(* IEC 61131-3 sources: POMIRTS_lab3/AS/Library/AsARCfg, 3 files *)

(* ---- AsARCfg.typ ---- *)
(********************************************************************
 * COPYRIGHT -- Bernecker + Rainer
 ********************************************************************
 * Library: AsARCfg
 * File: AsARCfg.typ
 * Author: B+R
 ********************************************************************
 * Data types of library AsARCfg
 ********************************************************************)

 TYPE
	cfgLease_typ : STRUCT				(*lease structure*)
		name			: STRING[8];	(*name of lease (max 8)*)
		startAdr		: STRING[16];	(*start address of lease*)
		stopAdr			: STRING[16];	(*stop address of lease*)
		subnetMask		: STRING[16];	(*subnet mask of lease*)
		defaultGateway	: STRING[16];	(*default gateway of lease*)
		leaseTimeout	: DINT;			(*-1 for infinite timeout*)
	END_STRUCT;
END_TYPE

(* ---- AsARCfg.fun ---- *)
(********************************************************************
 * COPYRIGHT -- Bernecker + Rainer
 ********************************************************************
 * Library: AsARCfg
 * File: AsARCfg.fun
 * Author: B+R
 ********************************************************************
 * Functions and function blocks of library AsARCfg
 ********************************************************************)

FUNCTION_BLOCK CfgGetInaNode			(*reads the node number from the AR registry for a INA device; asynchronous execution*)
	VAR_INPUT
		enable			: BOOL;			(*enables execution*)
		pDevice			: UDINT;		(*INA device name given as pointer (syntax: SL<x>.SS<y>.IF<z>)*)
	END_VAR

	VAR_OUTPUT
		status			: UINT;			(*execution status: ERR_OK, ERR_FUB_ENABLE_FALSE, ERR_FUB_BUSY, 0xXXXX = see help*)
		InaNode			: USINT;		(*INA node number*)
	END_VAR

	VAR
        i_state			: UINT;			(*internal variable*)
		i_result		: UINT;			(*internal variable*)
        i_tmp			: UDINT;		(*internal variable*)
	END_VAR
END_FUNCTION_BLOCK

FUNCTION_BLOCK CfgSetInaNode			(*enters the node number into the AR registry for INA device; asynchronous execution*)
	VAR_INPUT
		enable			: BOOL;			(*enables execution*)
		pDevice			: UDINT;		(*INA device name given as pointer (syntax: SL<x>.SS<y>.IF<z>)*)
		InaNode			: USINT;		(*INA node number*)
		Option			: UDINT;		(*options: cfgOPTION_VOLATILE, cfgOPTION_NON_VOLATILE*)
	END_VAR

	VAR_OUTPUT
		status			: UINT;			(*execution status: ERR_OK, ERR_FUB_ENABLE_FALSE, ERR_FUB_BUSY, 0xXXXX = see help*)
	END_VAR

	VAR
        i_state			: UINT;			(*internal variable*)
		i_result		: UINT;			(*internal variable*)
        i_tmp			: UDINT;		(*internal variable*)
	END_VAR
END_FUNCTION_BLOCK

FUNCTION_BLOCK CfgGetIPAddr				(*reads IP address from the AR registry for Ethernet device; asynchronous execution*)
	VAR_INPUT
		enable			: BOOL;			(*enables execution*)
		pDevice			: UDINT;		(*INA device name given as pointer (syntax: SL<x>.SS<y>.IF<z>)*)
		pIPAddr			: UDINT;		(*IP address given as a pointer*)
		Len				: USINT;		(*length of the string (pIPAddr) -> ideally, Len = 16*)
	END_VAR

	VAR_OUTPUT
		status			: UINT;			(*execution status: ERR_OK, ERR_FUB_ENABLE_FALSE, ERR_FUB_BUSY, 0xXXXX = see help*)
	END_VAR

	VAR
        i_state			: UINT;			(*internal variable*)
		i_result		: UINT;			(*internal variable*)
        i_tmp			: UDINT;		(*internal variable*)
	END_VAR
END_FUNCTION_BLOCK

FUNCTION_BLOCK CfgSetIPAddr				(*enters IP address into the AR registry for Ethernet device; asynchronous execution*)
	VAR_INPUT
		enable			: BOOL;			(*enables execution*)
		pDevice			: UDINT;		(*INA device name given as pointer (syntax: SL<x>.SS<y>.IF<z>)*)
		pIPAddr			: UDINT;		(*IP address given as pointer, valid range "1.0.0.1" - "247.255.255.255"*)
		Option			: UDINT;		(*options:  cfgOPTION_VOLATILE, cfgOPTION_NON_VOLATILE*)
	END_VAR

	VAR_OUTPUT
		status			: UINT;			(*execution status: ERR_OK, ERR_FUB_ENABLE_FALSE, ERR_FUB_BUSY, 0xXXXX = see help*)
	END_VAR

	VAR
        i_state			: UINT;			(*internal variable*)
		i_result		: UINT;			(*internal variable*)
        i_tmp			: UDINT;		(*internal variable*)
	END_VAR
END_FUNCTION_BLOCK

FUNCTION_BLOCK CfgGetSubnetMask			(*reads subnet mask from the AR registry for Ethernet device; asynchronous execution*)
	VAR_INPUT
		enable			: BOOL;			(*enables execution*)
		pDevice			: UDINT;		(*INA device name given as pointer (syntax: SL<x>.SS<y>.IF<z>)*)
		pSubnetMask		: UDINT;		(*subnet mask*)
		Len				: USINT;		(*length of the string (pSubnetMask) -> ideally, Len = 16*)
	END_VAR

	VAR_OUTPUT
		status			: UINT;			(*execution status: ERR_OK, ERR_FUB_ENABLE_FALSE, ERR_FUB_BUSY, 0xXXXX = see help*)
	END_VAR

	VAR
		i_state			: UINT;			(*internal variable*)
		i_result		: UINT;			(*internal variable*)
        i_tmp			: UDINT;		(*internal variable*)
	END_VAR
END_FUNCTION_BLOCK

FUNCTION_BLOCK CfgSetSubnetMask			(*enters subnet mask into the AR registry for Ethernet device; asynchronous execution*)
	VAR_INPUT
		enable			: BOOL;			(*enables execution*)
		pDevice			: UDINT;		(*INA device name given as pointer (syntax: SL<x>.SS<y>.IF<z>)*)
		pSubnetMask		: UDINT;		(*subnet mask given as a pointer, valid range "1.0.0.1" - "255.255.255.254"*)
		Option			: UDINT;		(*options: cfgOPTION_VOLATILE, cfgOPTION_NON_VOLATILE*)
	END_VAR

	VAR_OUTPUT
		status			: UINT;			(*execution status: ERR_OK, ERR_FUB_ENABLE_FALSE, ERR_FUB_BUSY, 0xXXXX = see help*)
	END_VAR

	VAR
        i_state			: UINT;			(*internal variable*)
		i_result		: UINT;			(*internal variable*)
        i_tmp			: UDINT;		(*internal variable*)
	END_VAR
END_FUNCTION_BLOCK

FUNCTION_BLOCK CfgGetDefaultGateway		(*reads default gateway from AR registry for Ethernet device; asynchronous execution*)
	VAR_INPUT
		enable			: BOOL;			(*enables execution*)
		pDevice			: UDINT;		(*INA device name given as pointer (syntax: SL<x>.SS<y>.IF<z>)*)
		pGateway		: UDINT;		(*default gateway address given as pointer*)
		Len				: USINT;		(*length of the string (pGateway) -> ideally, Len = 16*)
	END_VAR

	VAR_OUTPUT
		status			: UINT;			(*execution status: ERR_OK, ERR_FUB_ENABLE_FALSE, ERR_FUB_BUSY, 0xXXXX = see help*)
	END_VAR

	VAR
        i_state			: UINT;			(*internal variable*)
		i_result		: UINT;			(*internal variable*)
        i_tmp			: UDINT;		(*internal variable*)
	END_VAR
END_FUNCTION_BLOCK

FUNCTION_BLOCK CfgSetDefaultGateway		(*enters default gateway into AR registry for Ethernet device; asynchronous execution*)
	VAR_INPUT
		enable			: BOOL;			(*enables execution*)
		pDevice			: UDINT;		(*INA device name given as pointer (syntax: SL<x>.SS<y>.IF<z>)*)
		pGateway		: UDINT;		(*default gateway address given as pointer, valid range "1.0.0.1" - "247.255.255.255"*)
		Option			: UDINT;		(*options: cfgOPTION_VOLATILE, cfgOPTION_NON_VOLATILE*)
	END_VAR

	VAR_OUTPUT
		status			: UINT;			(*execution status: ERR_OK, ERR_FUB_ENABLE_FALSE, ERR_FUB_BUSY, 0xXXXX = see help*)
	END_VAR

	VAR
        i_state			: UINT;			(*internal variable*)
		i_result		: UINT;			(*internal variable*)
        i_tmp			: UDINT;		(*internal variable*)
	END_VAR
END_FUNCTION_BLOCK

FUNCTION_BLOCK CfgGetBroadcastAddr		(*reads broadcast address from AR registry for Ethernet device; asynchronous execution*)
	VAR_INPUT
		enable			: BOOL;			(*enables execution*)
		pDevice			: UDINT;		(*INA device name given as pointer (syntax: SL<x>.SS<y>.IF<z>)*)
		pBroadcastAddr	: UDINT;		(*broadcast address given as a pointer*)
		Len				: USINT;		(*length of the string (pBroadcastAddr) -> ideally, Len = 16*)
	END_VAR

	VAR_OUTPUT
		status			: UINT;			(*execution status: ERR_OK, ERR_FUB_ENABLE_FALSE, ERR_FUB_BUSY, 0xXXXX = see help*)
	END_VAR

	VAR
        i_state			: UINT;			(*internal variable*)
		i_result		: UINT;			(*internal variable*)
        i_tmp			: UDINT;		(*internal variable*)
	END_VAR
END_FUNCTION_BLOCK

FUNCTION_BLOCK CfgSetBroadcastAddr		(*enters broadcast address into the AR registry for Ethernet device; asynchronous execution*)
	VAR_INPUT
		enable			: BOOL;			(*enables execution*)
		pDevice			: UDINT;		(*INA device name given as pointer (syntax: SL<x>.SS<y>.IF<z>)*)
		pBroadcastAddr	: UDINT;		(*broadcast address given as a pointer, valid range "1.0.0.1" - "255.255.255.255"*)
		Option			: UDINT;		(*options: cfgOPTION_VOLATILE, cfgOPTION_NON_VOLATILE*)
	END_VAR

	VAR_OUTPUT
		status			: UINT;			(*execution status: ERR_OK, ERR_FUB_ENABLE_FALSE, ERR_FUB_BUSY, 0xXXXX = see help*)
	END_VAR

	VAR
        i_state			: UINT;			(*internal variable*)
		i_result		: UINT;			(*internal variable*)
        i_tmp			: UDINT;		(*internal variable*)
	END_VAR
END_FUNCTION_BLOCK

FUNCTION_BLOCK CfgGetEthBaudrate		(*reads the baud rate from the AR registry for Ethernet device; asynchronous execution*)
	VAR_INPUT
		enable			: BOOL;			(*enables execution*)
		pDevice			: UDINT;		(*INA device name given as pointer (syntax: SL<x>.SS<y>.IF<z>)*)
	END_VAR

	VAR_OUTPUT
		status			: UINT;			(*execution status: ERR_OK, ERR_FUB_ENABLE_FALSE, ERR_FUB_BUSY, 0xXXXX = see help*)
		Baudrate		: UDINT;		(*baud rate, e.g. cfgETHBAUDRATE_AUTO, cfgETHBAUDRATE_10, cfgETHBAUDRATE_10FD ...*)
	END_VAR

	VAR
        i_state			: UINT;			(*internal variable*)
		i_result		: UINT;			(*internal variable*)
        i_tmp			: UDINT;		(*internal variable*)
	END_VAR
END_FUNCTION_BLOCK

FUNCTION_BLOCK CfgSetEthBaudrate		(*enters the baud rate into the AR registry for Ethernet device; asynchronous execution*)
	VAR_INPUT
		enable			: BOOL;			(*enables execution*)
		pDevice			: UDINT;		(*INA device name given as pointer (syntax: SL<x>.SS<y>.IF<z>)*)
		Baudrate		: UDINT;		(*Ethernet baud rate, e.g. cfgETHBAUDRATE_AUTO, cfgETHBAUDRATE_10, cfgETHBAUDRATE_10FD ...*)
		Option			: UDINT;		(*options: cfgOPTION_VOLATILE, cfgOPTION_NON_VOLATILE*)
	END_VAR

	VAR_OUTPUT
		status			: UINT;			(*execution status: ERR_OK, ERR_FUB_ENABLE_FALSE, ERR_FUB_BUSY, 0xXXXX = see help*)
	END_VAR

	VAR
        i_state			: UINT;			(*internal variable*)
		i_result		: UINT;			(*internal variable*)
        i_tmp			: UDINT;		(*internal variable*)
	END_VAR
END_FUNCTION_BLOCK

FUNCTION_BLOCK CfgGetEthConfigMode		(*reads the configuration mode; asynchronous execution*)
	VAR_INPUT
		enable			: BOOL;			(*enables execution*)
		pDevice			: UDINT;		(*INA device name given as pointer (syntax: SL<x>.SS<y>.IF<z>)*)
	END_VAR

	VAR_OUTPUT
		status			: UINT;			(*execution status: ERR_OK, ERR_FUB_ENABLE_FALSE, ERR_FUB_BUSY, 0xXXXX = see help*)
		ConfigMode		: UDINT;		(*configuration mode: cfgCONFIGMODE_MANUALLY, cfgCONFIGMODE_DHCPCLIENT*)
	END_VAR

	VAR
        i_state			: UINT;			(*internal variable*)
		i_result		: UINT;			(*internal variable*)
        i_tmp			: UDINT;		(*internal variable*)
	END_VAR
END_FUNCTION_BLOCK

FUNCTION_BLOCK CfgSetEthConfigMode		(*modifies the configuration mode for Ethernet device; asynchronous execution*)
	VAR_INPUT
		enable			: BOOL;			(*enables execution*)
		pDevice			: UDINT;		(*INA device name given as pointer (syntax: SL<x>.SS<y>.IF<z>)*)
		ConfigMode		: UDINT;		(*configuration mode: cfgCONFIGMODE_MANUALLY, cfgCONFIGMODE_DHCPCLIENT*)
		Option			: UDINT;		(*options: cfgOPTION_VOLATILE, cfgOPTION_NON_VOLATILE*)
	END_VAR

	VAR_OUTPUT
		status			: UINT;			(*execution status: ERR_OK, ERR_FUB_ENABLE_FALSE, ERR_FUB_BUSY, 0xXXXX = see help*)
	END_VAR

	VAR
        i_state			: UINT;			(*internal variable*)
		i_result		: UINT;			(*internal variable*)
        i_tmp			: UDINT;		(*internal variable*)
	END_VAR
END_FUNCTION_BLOCK

FUNCTION_BLOCK CfgGetHostName			(*reads a host name for a target; asynchronous execution*)
	VAR_INPUT
		enable			: BOOL;			(*enables execution*)
		pHostName		: UDINT;		(*hostname*)
		Len				: USINT;		(*length of the string (HostName)*)
	END_VAR

	VAR_OUTPUT
		status			: UINT;			(*execution status: ERR_OK, ERR_FUB_ENABLE_FALSE, ERR_FUB_BUSY, 0xXXXX = see help*)
	END_VAR

	VAR
        i_state			: UINT;			(*internal variable*)
		i_result		: UINT;			(*internal variable*)
        i_tmp			: UDINT;		(*internal variable*)
	END_VAR
END_FUNCTION_BLOCK

FUNCTION_BLOCK CfgSetHostName			(*sets a host name for a target; asynchronous execution*)
	VAR_INPUT
		enable			: BOOL;			(*enables execution*)
		pHostName		: UDINT;		(*hostname*)
		Option			: UDINT;		(*options: cfgOPTION_VOLATILE, cfgOPTION_NON_VOLATILE*)
	END_VAR

	VAR_OUTPUT
		status			: UINT;			(*execution status: ERR_OK, ERR_FUB_ENABLE_FALSE, ERR_FUB_BUSY, 0xXXXX = see help*)
	END_VAR

	VAR
        i_state			: UINT;			(*internal variable*)
		i_result		: UINT;			(*internal variable*)
        i_tmp			: UDINT;		(*internal variable*)
	END_VAR
END_FUNCTION_BLOCK

FUNCTION_BLOCK CfgGetMacAddr			(*reads the MAC address of an Ethernet device*)
	VAR_INPUT
		enable			: BOOL;			(*enables execution*)
		pDevice			: UDINT;		(*INA device name given as pointer (syntax: SL<x>.SS<y>.IF<z>)*)
		pMacAddr		: UDINT;		(*MAC address (pointer to buffer where the MAC address should be written)*)
		Len				: USINT;		(*length of the MAC address (buffer - pMacAddr) -> normally 6 bytes*)
	END_VAR

	VAR_OUTPUT
		status			: UINT;			(*execution status: ERR_OK, ERR_FUB_ENABLE_FALSE, 0xXXXX = see help*)
	END_VAR

	VAR
        i_state			: UINT;			(*internal variable*)
		i_result		: UINT;			(*internal variable*)
        i_tmp			: UDINT;		(*internal variable*)
	END_VAR
END_FUNCTION_BLOCK

FUNCTION_BLOCK CfgSetFTPServer			(*enables/disables the FTP server*)
	VAR_INPUT
		enable			: BOOL;			(*enables execution*)
		Option			: UDINT;		(*options: cfgOPTION_DISABLE, cfgOPTION_ENABLE*)
	END_VAR

	VAR_OUTPUT
		status			: UINT;			(*execution status: ERR_OK, ERR_FUB_ENABLE_FALSE, 0xXXXX = see help*)
	END_VAR

	VAR
        i_state			: UINT;			(*internal variable*)
		i_result		: UINT;			(*internal variable*)
        i_tmp			: UDINT;		(*internal variable*)
	END_VAR
END_FUNCTION_BLOCK

FUNCTION_BLOCK CfgGetTimeOffset			(*returns the configured time offset*)
	VAR_INPUT
		enable			: BOOL;			(*enables execution*)
	END_VAR

	VAR_OUTPUT
		status			: UINT;			(*execution status: ERR_OK, ERR_FUB_ENABLE_FALSE, 0xXXXX = see help*)
		timeoffset		: INT;			(*configured time offset*)
	END_VAR

	VAR
        i_state			: UINT;			(*internal variable*)
		i_result		: UINT;			(*internal variable*)
        i_tmp			: UDINT;		(*internal variable*)
	END_VAR
END_FUNCTION_BLOCK

FUNCTION_BLOCK CfgSetTimeOffset			(*sets a time offset*)
	VAR_INPUT
		enable			: BOOL;			(*enables execution*)
        timeoffset		: INT;			(*configured time offset*)
        option			: UDINT;		(*options: cfgOPTION_VOLATILE, cfgOPTION_NON_VOLATILE*)
	END_VAR

	VAR_OUTPUT
        status			: UINT;			(*execution status: ERR_OK, ERR_FUB_ENABLE_FALSE, 0xXXXX = see help*)
	END_VAR

	VAR
        i_state			: UINT;			(*internal variable*)
		i_result		: UINT;			(*internal variable*)
        i_tmp			: UDINT;		(*internal variable*)
	END_VAR
END_FUNCTION_BLOCK

FUNCTION_BLOCK CfgSetSntpServer			(*starts the SNTP server*)
	VAR_INPUT
		enable			: BOOL;			(*enables execution*)
        start			: UDINT;		(*1 Starts the SNTP server*)
        option			: UDINT;		(*Options: cfgOPTION_VOLATILE, cfgOPTION_NON_VOLATILE*)
	END_VAR

	VAR_OUTPUT
        status			: UINT;			(*execution status: ERR_OK, ERR_FUB_ENABLE_FALSE, 0xXXXX = see help*)
	END_VAR

	VAR
        i_state			: UINT;			(*internal variable*)
		i_result		: UINT;			(*internal variable*)
        i_tmp			: UDINT;		(*internal variable*)
	END_VAR
END_FUNCTION_BLOCK

FUNCTION_BLOCK CfgSetSntpClient			(*starts and stops the SNTP client*)
	VAR_INPUT
		enable			: BOOL;			(*enables execution*)
		run				: UDINT;		(*0 stop client, 1 start client*)
		pServerAddr		: UDINT;		(*pointer to a string with the IP address of the SNTP server*)
		sntpcInterval	: UINT;			(*interval in minutes that it takes for the SNTP client to synchronize the time with the server*)
		rtcInterval		: UINT;			(*interval in minutes that it takes to synchronize the RTC with the software time during SNTP operation*)
		option			: UDINT;		(*options: cfgOPTION_VOLATILE, cfgOPTION_NON_VOLATILE*)
	END_VAR

	VAR_OUTPUT
		status			: UINT;			(*execution status: ERR_OK, ERR_FUB_ENABLE_FALSE, 0xXXXX = see help*)
		syncStatus		: USINT;		(*0 Client not active, 1 Client already active, but time not received from server, ...*)
	END_VAR

	VAR
        i_state			: UINT;			(*internal variable*)
		i_result		: UINT;			(*internal variable*)
        i_tmp			: UDINT;		(*internal variable*)
	END_VAR
END_FUNCTION_BLOCK

FUNCTION_BLOCK CfgGetSntpcData			(*returns the parameters relevant for the SNTP client*)
	VAR_INPUT
		enable			: BOOL;			(*enables execution*)
		pServerAddr		: UDINT;		(*pointer to a long enough string to contain the server address or server name*)
		Len				: USINT;		(*length of the string (pServerAddr)*)
	END_VAR

	VAR_OUTPUT
		status			: UINT;			(*execution status: ERR_OK, ERR_FUB_ENABLE_FALSE, 0xXXXX = see help*)
		run				: UDINT;		(*1 Client active, 0 Client inactive*)
        sntpcInterval	: UINT;			(*interval that it takes for the SNTP client to synchronize the time with the server*)
        rtcInterval		: UINT;			(*interval that it take to synchronize the RTC with the software time during SNTP operation*)
	END_VAR

	VAR
        i_state			: UINT;			(*internal variable*)
		i_result		: UINT;			(*internal variable*)
        i_tmp			: UDINT;		(*internal variable*)
	END_VAR
END_FUNCTION_BLOCK

FUNCTION_BLOCK CfgGetSntpsData			(*returns whether the SNTP server is active*)
	VAR_INPUT
		enable			: BOOL;			(*enables execution*)
	END_VAR

	VAR_OUTPUT
		status			: UINT;			(*execution status: ERR_OK, ERR_FUB_ENABLE_FALSE, 0xXXXX = see help*)
		run				: UDINT;		(*1 server active, 0 server inactive*)
	END_VAR

	VAR
        i_state			: UINT;			(*internal variable*)
		i_result		: UINT;			(*internal variable*)
        i_tmp			: UDINT;		(*internal variable*)
	END_VAR
END_FUNCTION_BLOCK

FUNCTION_BLOCK CfgGetTimeZone
	VAR_INPUT
		enable			: BOOL;			(*enables execution*)
	END_VAR

	VAR_OUTPUT
		timezoneID		: UINT;
        status			: UINT;			(*execution status: ERR_OK, ERR_FUB_ENABLE_FALSE, ERR_FUB_BUSY, 0xXXXX = see help*)
	END_VAR

	VAR
        i_state			: UINT;			(*internal variable*)
		i_result		: UINT;			(*internal variable*)
        i_tmp			: UDINT;		(*internal variable*)
	END_VAR
END_FUNCTION_BLOCK

FUNCTION_BLOCK CfgSetTimeZone
	VAR_INPUT
		enable			: BOOL;			(*enables execution*)
		timezoneID		: UINT;
		option			: UDINT;
	END_VAR

	VAR_OUTPUT
        status			: UINT;			(*execution status: ERR_OK, ERR_FUB_ENABLE_FALSE, ERR_FUB_BUSY, 0xXXXX = see help*)
	END_VAR

	VAR
        i_state			: UINT;			(*internal variable*)
		i_result		: UINT;			(*internal variable*)
        i_tmp			: UDINT;		(*internal variable*)
	END_VAR
END_FUNCTION_BLOCK

FUNCTION_BLOCK CfgGetTimeZoneInfo
	VAR_INPUT
		enable			: BOOL;			(*enables execution*)
		timezoneID		: UINT;
	END_VAR

	VAR_OUTPUT
		gmt				: INT;
		gmtDst			: INT;
        status			: UINT;			(*execution status: ERR_OK, ERR_FUB_ENABLE_FALSE, ERR_FUB_BUSY, 0xXXXX = see help*)
	END_VAR

	VAR
        i_state			: UINT;			(*internal variable*)
		i_result		: UINT;			(*internal variable*)
        i_tmp			: UDINT;		(*internal variable*)
	END_VAR
END_FUNCTION_BLOCK

FUNCTION_BLOCK CfgGetTimeZoneEntry
	VAR_INPUT
		enable			: BOOL;			(*enables execution*)
		timezoneID		: UINT;
		year			: UINT;
	END_VAR

	VAR_OUTPUT
		dateDst			: DATE_AND_TIME;
		dateNormal		: DATE_AND_TIME;
        status			: UINT;			(*execution status: ERR_OK, ERR_FUB_ENABLE_FALSE, ERR_FUB_BUSY, 0xXXXX = see help*)
	END_VAR

	VAR
        i_state			: UINT;			(*internal variable*)
		i_result		: UINT;			(*internal variable*)
        i_tmp			: UDINT;		(*internal variable*)
	END_VAR
END_FUNCTION_BLOCK

FUNCTION_BLOCK CfgGetDst
	VAR_INPUT
		enable			: BOOL;			(*enables execution*)
	END_VAR

	VAR_OUTPUT
		dst				: BOOL;
        status			: UINT;			(*execution status: ERR_OK, ERR_FUB_ENABLE_FALSE, ERR_FUB_BUSY, 0xXXXX = see help*)
	END_VAR

	VAR
        i_state			: UINT;			(*internal variable*)
		i_result		: UINT;			(*internal variable*)
        i_tmp			: UDINT;		(*internal variable*)
	END_VAR
END_FUNCTION_BLOCK

FUNCTION_BLOCK CfgSetDst
	VAR_INPUT
		enable			: BOOL;			(*enables execution*)
		dst				: BOOL;
		option			: UDINT;
	END_VAR

	VAR_OUTPUT
        status			: UINT;			(*execution status: ERR_OK, ERR_FUB_ENABLE_FALSE, ERR_FUB_BUSY, 0xXXXX = see help*)
	END_VAR

	VAR
        i_state			: UINT;			(*internal variable*)
		i_result		: UINT;			(*internal variable*)
        i_tmp			: UDINT;		(*internal variable*)
	END_VAR
END_FUNCTION_BLOCK

FUNCTION_BLOCK CfgGetCIFSDomain				(*cifs - reads domain name from the AR registry; asynchronous execution*)
	VAR_INPUT
		enable			: BOOL;			(*enables execution*)
		pDomain			: UDINT;		(*Domainname given as a pointer*)
		Len				: USINT;		(*length of the string (pDomain) -> ideally, Len = 16*)
	END_VAR

	VAR_OUTPUT
		isWorkgroup		: USINT;		(*specifies if Workgroup or Domain*)
		status			: UINT;			(*execution status: ERR_OK, ERR_FUB_ENABLE_FALSE, ERR_FUB_BUSY, 0xXXXX = see help*)
	END_VAR

	VAR
        i_state			: UINT;			(*internal variable*)
		i_result		: UINT;			(*internal variable*)
        i_tmp			: UDINT;		(*internal variable*)
	END_VAR
END_FUNCTION_BLOCK

FUNCTION_BLOCK CfgSetCIFSDomain			(*cifs - enters domain into the AR registry; asynchronous execution*)
	VAR_INPUT
		enable			: BOOL;			(*enables execution*)
		pDomain			: UDINT;		(*Domainname given as pointer*)
		isWorkgroup		: USINT;		(*specifies if Workgroup or Domain cfgOPTION_NON_WORKGROUP, cfgOPTION_WORKGROUP*)
		Option			: UDINT;		(*options:  cfgOPTION_VOLATILE, cfgOPTION_NON_VOLATILE*)
	END_VAR

	VAR_OUTPUT
		status			: UINT;			(*execution status: ERR_OK, ERR_FUB_ENABLE_FALSE, ERR_FUB_BUSY, 0xXXXX = see help*)
	END_VAR

	VAR
        i_state			: UINT;			(*internal variable*)
		i_result		: UINT;			(*internal variable*)
        i_tmp			: UDINT;		(*internal variable*)
	END_VAR
END_FUNCTION_BLOCK

FUNCTION_BLOCK CfgGetCIFSDefaultuser	(*cifs - reads default user from the AR registry; asynchronous execution*)
	VAR_INPUT
		enable				: BOOL;			(*enables execution*)
		pDefaultuser		: UDINT;		(*Default Username given as a pointer*)
		lenUser				: USINT;		(*length of the string (pDefaultuser) -> ideally, Len = 16*)
		pDefaultpassword	: UDINT;		(*Default Password given as a pointer*)
		lenPassword			: USINT;		(*length of the string (pDefaultpassword) -> ideally, Len = 16*)
	END_VAR

	VAR_OUTPUT
		status			: UINT;			(*execution status: ERR_OK, ERR_FUB_ENABLE_FALSE, ERR_FUB_BUSY, 0xXXXX = see help*)
	END_VAR

	VAR
        i_state			: UINT;			(*internal variable*)
		i_result		: UINT;			(*internal variable*)
        i_tmp			: UDINT;		(*internal variable*)
	END_VAR
END_FUNCTION_BLOCK

FUNCTION_BLOCK CfgSetCIFSDefaultuser	(*cifs - enters default user into the AR registry; asynchronous execution*)
	VAR_INPUT
		enable				: BOOL;			(*enables execution*)
		pDefaultuser		: UDINT;		(*Default Username given as pointer*)
		pDefaultpassword	: UDINT;		(*Default Password given as a pointer*)
		Option				: UDINT;		(*options:  cfgOPTION_VOLATILE, cfgOPTION_NON_VOLATILE*)
	END_VAR

	VAR_OUTPUT
		status			: UINT;			(*execution status: ERR_OK, ERR_FUB_ENABLE_FALSE, ERR_FUB_BUSY, 0xXXXX = see help*)
	END_VAR

	VAR
        i_state			: UINT;			(*internal variable*)
		i_result		: UINT;			(*internal variable*)
        i_tmp			: UDINT;		(*internal variable*)
	END_VAR
END_FUNCTION_BLOCK

FUNCTION_BLOCK CfgSetDhcpServer 	(*dhcp - starts or stops dhcp server*)
	VAR_INPUT
		enable				: BOOL;			(*enables execution*)
		start				: UDINT;		(*1 = start server; 0 = stop server*)
		option				: UDINT;		(*options:  cfgOPTION_VOLATILE, cfgOPTION_NON_VOLATILE*)
	END_VAR

	VAR_OUTPUT
		status			: UINT;			(*execution status: ERR_OK, ERR_FUB_ENABLE_FALSE, ERR_FUB_BUSY, 0xXXXX = see help*)
	END_VAR

	VAR
        i_state			: UINT;			(*internal variable*)
		i_result		: UINT;			(*internal variable*)
        i_tmp			: UDINT;		(*internal variable*)
	END_VAR
END_FUNCTION_BLOCK

FUNCTION_BLOCK CfgSetDhcpsData 	(*dhcp - configures dhcp server*)
	VAR_INPUT
		enable				: BOOL;			(*enables execution*)
		pInterfaceList		: UDINT;		(*provided interfaces*)
		pLeases				: UDINT;		(*provided leases*)
		numLeases			: UDINT;		(*number of leases*)
		option				: UDINT;		(*options:  cfgOPTION_VOLATILE, cfgOPTION_NON_VOLATILE*)
	END_VAR

	VAR_OUTPUT
		status			: UINT;			(*execution status: ERR_OK, ERR_FUB_ENABLE_FALSE, ERR_FUB_BUSY, 0xXXXX = see help*)
	END_VAR

	VAR
        i_state			: UINT;			(*internal variable*)
		i_result		: UINT;			(*internal variable*)
        i_tmp			: UDINT;		(*internal variable*)
	END_VAR
END_FUNCTION_BLOCK

FUNCTION_BLOCK CfgGetDhcpsData 	(*dhcp - reads configuration of dhcp server*)
	VAR_INPUT
		enable				: BOOL;			(*enables execution*)
		pInterfaceList		: UDINT;		(*provided interfaces*)
		len					: UDINT;		(*length of the string (pInterfaces)*)
		pLeases				: UDINT;		(*provided leases*)
		numLeases			: UDINT;		(*number of leases*)
	END_VAR

	VAR_OUTPUT
		startMode		: UDINT;		(*1 = server is working; 0 = server is not working*)
		numNeeded		: UDINT;		(*needed length*)
		status			: UINT;			(*execution status: ERR_OK, ERR_FUB_ENABLE_FALSE, ERR_FUB_BUSY, 0xXXXX = see help*)
	END_VAR

	VAR
        i_state			: UINT;			(*internal variable*)
		i_result		: UINT;			(*internal variable*)
        i_tmp			: UDINT;		(*internal variable*)
	END_VAR
END_FUNCTION_BLOCK

FUNCTION_BLOCK CfgSetSdmStatus			(*enables/disables data refresh of system diagnostics manager*)
	VAR_INPUT
		enable			: BOOL;			(*enables execution*)
		start			: UDINT;		(*options: cfgOPTION_ENABLE_SDM; cfgOPTION_DISABLE_SDM*)
		Option			: UDINT;		(*reserve*)
	END_VAR

	VAR_OUTPUT
		status			: UINT;			(*execution status: ERR_OK, ERR_FUB_ENABLE_FALSE, 0xXXXX = see help*)
	END_VAR

	VAR
        i_state			: UINT;			(*internal variable*)
		i_result		: UINT;			(*internal variable*)
        i_tmp			: UDINT;		(*internal variable*)
	END_VAR
END_FUNCTION_BLOCK

FUNCTION_BLOCK CfgGetSdmStatus			(*returns whether the system diagnostics manager is active*)
	VAR_INPUT
		enable			: BOOL;			(*enables execution*)
	END_VAR

	VAR_OUTPUT
		status			: UINT;			(*execution status: ERR_OK, ERR_FUB_ENABLE_FALSE, 0xXXXX = see help*)
		run				: UDINT;		(*status: cfgSTATUS_SDM_ENABLED, cfgSTATUS_SDM_DISABLED*)
	END_VAR

	VAR
        i_state			: UINT;			(*internal variable*)
		i_result		: UINT;			(*internal variable*)
        i_tmp			: UDINT;		(*internal variable*)
	END_VAR
END_FUNCTION_BLOCK

FUNCTION CfgClearNV		: UINT			(*clear non volatile data*)
END_FUNCTION

FUNCTION_BLOCK CfgSetSdmColor			(*set the system diagnostics manager color scheme*)
	VAR_INPUT
		enable			: BOOL;			(*enables execution*)
		red  			: UDINT;  		(*red value (0-255)*)
		green  			: UDINT;  		(*green value (0-255)*)
		blue  			: UDINT;  		(*blue value (0-255)*)
		Option			: UDINT;		(*options: cfgOPTION_VOLATILE, cfgOPTION_NON_VOLATILE*)
	END_VAR

	VAR_OUTPUT
		status			: UINT;			(*execution status: ERR_OK, ERR_FUB_ENABLE_FALSE, 0xXXXX = see help*)
	END_VAR

	VAR
        i_state			: UINT;			(*internal variable*)
		i_result		: UINT;			(*internal variable*)
        i_tmp			: UDINT;		(*internal variable*)
	END_VAR
END_FUNCTION_BLOCK

FUNCTION_BLOCK CfgGetSdmColor			(*get the system diagnostics manager color scheme*)
	VAR_INPUT
		enable			: BOOL;			(*enables execution*)
	END_VAR

	VAR_OUTPUT
		status			: UINT;			(*execution status: ERR_OK, ERR_FUB_ENABLE_FALSE, 0xXXXX = see help*)
		red  			: UDINT;  		(*red value (0-255)*)
		green  			: UDINT;  		(*green value (0-255)*)
		blue  			: UDINT;  		(*blue value (0-255)*)
	END_VAR

	VAR
        i_state			: UINT;			(*internal variable*)
		i_result		: UINT;			(*internal variable*)
        i_tmp			: UDINT;		(*internal variable*)
	END_VAR
END_FUNCTION_BLOCK

FUNCTION_BLOCK CfgGetSdmCustomData1 	(*sdm - get custom data 1 *)
	VAR_INPUT
		enable			: BOOL;			(*enables execution*)
		pDevice			: UDINT;		(*Devicename given as a pointer*)
		lenDevice		: UDINT;		(*length of the string (pDevice) -> ideally, Len = 255*)
		pFile			: UDINT;		(*Filename given as a pointer*)
		lenFile			: UDINT;		(*length of the string (pFile) -> ideally, Len = 255*)
		pDatamodule		: UDINT;		(*Datamodulename given as a pointer*)
		lenDatamodule	: UDINT;		(*length of the string (pDatamodule) -> ideally, Len = 255*)
	END_VAR

	VAR_OUTPUT
		status			: UINT;			(*execution status: ERR_OK, ERR_FUB_ENABLE_FALSE, ERR_FUB_BUSY, 0xXXXX = see help*)
	END_VAR

	VAR
        i_state			: UINT;			(*internal variable*)
		i_result		: UINT;			(*internal variable*)
        i_tmp			: UDINT;		(*internal variable*)
	END_VAR
END_FUNCTION_BLOCK

FUNCTION_BLOCK CfgSetSdmCustomData1 	(*sdm - set custom data 1 *)
	VAR_INPUT
		enable			: BOOL;			(*enables execution*)
		pDevice			: UDINT;		(*Devicename given as a pointer*)
		pFile			: UDINT;		(*Filename given as a pointer*)
		pDatamodule		: UDINT;		(*Datamodulename given as a pointer*)
		Option			: UDINT;		(*options: cfgOPTION_VOLATILE, cfgOPTION_NON_VOLATILE*)
	END_VAR

	VAR_OUTPUT
		status			: UINT;			(*execution status: ERR_OK, ERR_FUB_ENABLE_FALSE, ERR_FUB_BUSY, 0xXXXX = see help*)
	END_VAR

	VAR
        i_state			: UINT;			(*internal variable*)
		i_result		: UINT;			(*internal variable*)
        i_tmp			: UDINT;		(*internal variable*)
	END_VAR
END_FUNCTION_BLOCK

FUNCTION_BLOCK CfgGetSdmCustomData2 	(*sdm - get custom data 2 *)
	VAR_INPUT
		enable			: BOOL;			(*enables execution*)
		pDevice			: UDINT;		(*Devicename given as a pointer*)
		lenDevice		: UDINT;		(*length of the string (pDevice) -> ideally, Len = 255*)
		pFile			: UDINT;		(*Filename given as a pointer*)
		lenFile			: UDINT;		(*length of the string (pFile) -> ideally, Len = 255*)
		pDatamodule		: UDINT;		(*Datamodulename given as a pointer*)
		lenDatamodule	: UDINT;		(*length of the string (pDatamodule) -> ideally, Len = 255*)
	END_VAR

	VAR_OUTPUT
		status			: UINT;			(*execution status: ERR_OK, ERR_FUB_ENABLE_FALSE, ERR_FUB_BUSY, 0xXXXX = see help*)
	END_VAR

	VAR
        i_state			: UINT;			(*internal variable*)
		i_result		: UINT;			(*internal variable*)
        i_tmp			: UDINT;		(*internal variable*)
	END_VAR
END_FUNCTION_BLOCK

FUNCTION_BLOCK CfgSetSdmCustomData2 	(*sdm - set custom data 2 *)
	VAR_INPUT
		enable			: BOOL;			(*enables execution*)
		pDevice			: UDINT;		(*Devicename given as a pointer*)
		pFile			: UDINT;		(*Filename given as a pointer*)
		pDatamodule		: UDINT;		(*Datamodulename given as a pointer*)
		Option			: UDINT;		(*options: cfgOPTION_VOLATILE, cfgOPTION_NON_VOLATILE*)
	END_VAR

	VAR_OUTPUT
		status			: UINT;			(*execution status: ERR_OK, ERR_FUB_ENABLE_FALSE, ERR_FUB_BUSY, 0xXXXX = see help*)
	END_VAR

	VAR
        i_state			: UINT;			(*internal variable*)
		i_result		: UINT;			(*internal variable*)
        i_tmp			: UDINT;		(*internal variable*)
	END_VAR
END_FUNCTION_BLOCK

FUNCTION_BLOCK CfgGetWebMimeType 	(*webserver - set mime type *)
	VAR_INPUT
		enable			: BOOL;			(*enables execution*)
		pFileExtension	: UDINT;		(*Fileextension gives a pointer*)
		pMimeType		: UDINT;		(*MimeType given as a pointer*)
		len				: UDINT;		(*length of the string (pMimeType) -> ideally, Len = 255*)
	END_VAR

	VAR_OUTPUT
		status			: UINT;			(*execution status: ERR_OK, ERR_FUB_ENABLE_FALSE, ERR_FUB_BUSY, 0xXXXX = see help*)
	END_VAR

	VAR
        i_state			: UINT;			(*internal variable*)
		i_result		: UINT;			(*internal variable*)
        i_tmp			: UDINT;		(*internal variable*)
	END_VAR
END_FUNCTION_BLOCK

FUNCTION_BLOCK CfgSetWebMimeType 	(*webserver - get mime type*)
	VAR_INPUT
		enable			: BOOL;			(*enables execution*)
		mode			: BOOL;			(*cfgWEB_MODE_MIME_DEL(0) or cfgWEB_MODE_MIME_ADD(1)*)
		pFileExtension	: UDINT;		(*Fileextension gives a pointer*)
		pMimeType		: UDINT;		(*MimeType given as a pointer*)
		Option			: UDINT;		(*options: cfgOPTION_VOLATILE, cfgOPTION_NON_VOLATILE*)
	END_VAR

	VAR_OUTPUT
		status			: UINT;			(*execution status: ERR_OK, ERR_FUB_ENABLE_FALSE, ERR_FUB_BUSY, 0xXXXX = see help*)
	END_VAR

	VAR
        i_state			: UINT;			(*internal variable*)
		i_result		: UINT;			(*internal variable*)
        i_tmp			: UDINT;		(*internal variable*)
	END_VAR
END_FUNCTION_BLOCK

FUNCTION_BLOCK CfgGetWebServerPort 	(*webserver - get port number*)
	VAR_INPUT
		enable			: BOOL;			(*enables execution*)
	END_VAR

	VAR_OUTPUT
		status			: UINT;			(*execution status: ERR_OK, ERR_FUB_ENABLE_FALSE, ERR_FUB_BUSY, 0xXXXX = see help*)
		port  			: UINT;  		(*port number*)
	END_VAR

	VAR
        i_state			: UINT;			(*internal variable*)
		i_result		: UINT;			(*internal variable*)
        i_tmp			: UDINT;		(*internal variable*)
	END_VAR
END_FUNCTION_BLOCK

FUNCTION_BLOCK CfgGetWebServerDevice 	(*webserver - get webserver root directory*)
	VAR_INPUT
		enable			: BOOL;			(*enables execution*)
		pDevice 		: UDINT;  		(*Root directory name given as pointer*)
		len				: UDINT;		(*length of the string (pDevice) -> ideally, Len = 255*)
	END_VAR

	VAR_OUTPUT
		status			: UINT;			(*execution status: ERR_OK, ERR_FUB_ENABLE_FALSE, ERR_FUB_BUSY, 0xXXXX = see help*)
	END_VAR

	VAR
        i_state			: UINT;			(*internal variable*)
		i_result		: UINT;			(*internal variable*)
        i_tmp			: UDINT;		(*internal variable*)
	END_VAR
END_FUNCTION_BLOCK

FUNCTION_BLOCK CfgGetWebAspGoform 	(*webserver - get webserver ASP form*)
	VAR_INPUT
		enable			: BOOL;			(*enables execution*)
	END_VAR

	VAR_OUTPUT
		status			: UINT;			(*execution status: ERR_OK, ERR_FUB_ENABLE_FALSE, ERR_FUB_BUSY, 0xXXXX = see help*)
		mode			: UINT;			(*webserver - get webserver ASP form*)
	END_VAR

	VAR
        i_state			: UINT;			(*internal variable*)
		i_result		: UINT;			(*internal variable*)
        i_tmp			: UDINT;		(*internal variable*)
	END_VAR
END_FUNCTION_BLOCK

FUNCTION_BLOCK CfgSetWebAspGoform 	(*webserver - set webserver ASP form*)
	VAR_INPUT
		enable			: BOOL;			(*enables execution*)
		mode			: UINT;			(*webserver - set webserver ASP form*)
		Option			: UDINT;		(*options: cfgOPTION_VOLATILE, cfgOPTION_NON_VOLATILE*)
	END_VAR

	VAR_OUTPUT
		status			: UINT;			(*execution status: ERR_OK, ERR_FUB_ENABLE_FALSE, ERR_FUB_BUSY, 0xXXXX = see help*)
	END_VAR

	VAR
        i_state			: UINT;			(*internal variable*)
		i_result		: UINT;			(*internal variable*)
        i_tmp			: UDINT;		(*internal variable*)
	END_VAR
END_FUNCTION_BLOCK

FUNCTION_BLOCK CfgGetWebServerStatus 	(*webserver - get webserver status*)
	VAR_INPUT
		enable			: BOOL;			(*enables execution*)
	END_VAR

	VAR_OUTPUT
		status			: UINT;			(*execution status: ERR_OK, ERR_FUB_ENABLE_FALSE, ERR_FUB_BUSY, 0xXXXX = see help*)
		mode			: UINT;			(*cfgWEB_MODE_DISABLED(0) cfgWEB_MODE_ENABLED(1)*)
	END_VAR

	VAR
        i_state			: UINT;			(*internal variable*)
		i_result		: UINT;			(*internal variable*)
        i_tmp			: UDINT;		(*internal variable*)
	END_VAR
END_FUNCTION_BLOCK

FUNCTION_BLOCK CfgSetWebServerStatus 	(*webserver - set webserver status*)
	VAR_INPUT
		enable			: BOOL;			(*enables execution*)
		mode			: UINT;			(*cfgWEB_MODE_DISABLED(0) cfgWEB_MODE_ENABLED(1)*)
		Option			: UDINT;		(*options: cfgOPTION_VOLATILE, cfgOPTION_NON_VOLATILE*)
	END_VAR

	VAR_OUTPUT
		status			: UINT;			(*execution status: ERR_OK, ERR_FUB_ENABLE_FALSE, ERR_FUB_BUSY, 0xXXXX = see help*)
	END_VAR

	VAR
        i_state			: UINT;			(*internal variable*)
		i_result		: UINT;			(*internal variable*)
        i_tmp			: UDINT;		(*internal variable*)
	END_VAR
END_FUNCTION_BLOCK

(* ---- AsARCfg.var ---- *)
(********************************************************************
 * COPYRIGHT -- Bernecker + Rainer
 ********************************************************************
 * Library: AsARCfg
 * File: AsARCfg.var
 * Author: B+R
 ********************************************************************
 * Local variables of library AsARCfg
 ********************************************************************)

VAR CONSTANT
	cfgERR_DEVICE_NOT_EXIST			: UINT		:= 29000;	(*device doesn't exist or device not configured*)
	cfgERR_DEVICE_INVALID			: UINT		:= 29001;	(*FBK "pDevice" parameter invalid (e.g. pDevice = 0)*)
	cfgERR_OPTION_INVALID			: UINT		:= 29002;	(*FBK "Option" parameter invalid*)
	cfgERR_VALUE_INVALID			: UINT		:= 29003;	(*invalid FBK parameter, error text depends on the function block*)
	cfgERR_SET_NOT_POSSIBLE			: UINT		:= 29004;	(*not possible to set the subnet mask (e.g. DHCP client)*)
	cfgERR_ARREG					: UINT		:= 29005;	(*error in the AR registry*)
	cfgERR_INANODE_NOT_SUPPORTED	: UINT		:= 29006;	(*INA device does not support INA node numbers (e.g. IF1 = RS232)*)
	cfgERR_FTP_SINIT				: UINT		:= 29007;	(*initialization error on FTP server*)
	cfgERR_FTP_SDOWN				: UINT		:= 29008;	(*shutdown error on FTP server*)
	cfgERR_PARAM_NOT_SET			: UINT		:= 29009;	(*default gateway not defined*)
	cfgERR_SNTP_SERVER 				: UINT		:= 29010;	(*could not start the SNTP server*)
	cfgERR_SNTP_CLIENT 				: UINT		:= 29011;	(*error starting SNTP client (e.g. client already running)*)
	cfgERR_SNTP_INTERVAL 			: UINT		:= 29012;	(*invalid FBK parameter - values from 1 to 60 are valid*)
	cfgERR_SYSTEM		 			: UINT		:= 29013;	(*unexpected system error*)
	cfgERR_TIMEZONE					: UINT		:= 29014;   (*invalid timezone specified*)
	cfgERR_YEAR_INVALID				: UINT		:= 29015;	(*invalid year specified*)
	cfgERR_CIFS_DOMAIN_INVALID		: UINT 		:= 29016;   (*cifs domain name not defined *)
	cfgERR_CIFS_DEFAULTUSER_INVALID	: UINT		:= 29017;	(*cifs defaultuser not defined *)
	cfgERR_INANODE_NUMBER_SET       : UINT      := 29018;	(*could not set the INA node number*)
	cfgERR_CIFS_DEFAULTPW_INVALID	: UINT		:= 29019;	(*cifs default password not defined *)
	cfgERR_DHCP_SERVER_STARTED		: UINT		:= 29020;	(*server is already working*)
	cfgERR_INTERFACELIST_BUFFER		: UINT		:= 29021;	(*interfacelist buffer to small*)
	cfgERR_LEASES_BUFFER			: UINT		:= 29022;	(*leases array to small*)
	cfgERR_LEASE_EXISTS				: UINT		:= 29023;	(*leasename already exists*)
	cfgERR_LEASE_TIMEOUT			: UINT		:= 29024;	(*invalid lease timeout*)
	cfgERR_SDM_FUNCTION_NOT_FOUND	: UINT		:= 29026;	(*used arsdm function was not found*)
	cfgERR_CLEAR_NV_DATA			: UINT		:= 29027;	(*could not clear NV data*)
	cfgERR_FUNCTION_NOT_FOUND	    : UINT		:= 29028;	(*referenced function was not found*)
	cfgERR_SDM_DISABLED 		    : UINT      := 29029;	(*System diagnostics disabled*)
	cfgERR_WEBSERV_DISABLED 		: UINT      := 29030;	(*Web Server disabled*)

	cfgETHBAUDRATE_AUTO				: UDINT		:= 0;		(*auto-detect*)
	cfgETHBAUDRATE_10				: UDINT		:= 10;		(*10 MBaud, half-duplex*)
	cfgETHBAUDRATE_10FD				: UDINT		:= 11;		(*10 MBaud, full-duplex*)
	cfgETHBAUDRATE_100				: UDINT		:= 100;		(*100 MBaud, half-duplex*)
	cfgETHBAUDRATE_100FD			: UDINT		:= 101;		(*100 MBaud, full-duplex*)
	cfgETHBAUDRATE_1000FD			: UDINT		:= 1001;	(*1 GBaud, full-duplex*)

	cfgOPTION_NON_VOLATILE			: UDINT		:= 1;		(*permanently sets parameters*)
	cfgOPTION_VOLATILE				: UDINT		:= 0;		(*temporarily sets parameters*)

	cfgCONFIGMODE_MANUALLY			: UDINT		:= 0;		(*manual configuration*)
	cfgCONFIGMODE_DHCPCLIENT		: UDINT		:= 1;		(*DHCP client*)

	cfgOPTION_DISABLE				: UDINT		:= 0;		(*disable*)
	cfgOPTION_ENABLE				: UDINT		:= 1;		(*enable*)

	cfgOPTION_WORKGROUP				: USINT		:= 1;		(*Domain is Workgroup*)
	cfgOPTION_NON_WORKGROUP			: USINT		:= 0;		(*Domain isn't Workgroup*)

	cfgOPTION_ENABLE_SDM			: USINT		:= 1;		(*enable sdm*)
	cfgOPTION_DISABLE_SDM			: USINT		:= 2;		(*disable sdm*)

	cfgSTATUS_SDM_ENABLED			: USINT		:= 1;		(*sdm is enabled*)
	cfgSTATUS_SDM_DISABLED			: USINT		:= 2;		(*sdm is disabled*)

	cfgWEB_MODE_GOFORM_DISABLE		: UINT		:= 0;		(*Webserver Goform disabled*)
	cfgWEB_MODE_GOFORM_ENABLE		: UINT		:= 1;		(*Webserver Goform enabled*)
	cfgWEB_MODE_GOFORM_NO_WRITE		: UINT		:= 2;		(*Webserver Goform readonly*)

	cfgWEB_MODE_MIME_DEL			: UINT		:= 0;		(*Webserver delete MimeType*)
	cfgWEB_MODE_MIME_ADD			: UINT		:= 1;		(*Webserver set MimeType*)

	cfgWEB_MODE_DISABLED			: UINT		:= 0;		(*Webserver disabled*)
	cfgWEB_MODE_ENABLED				: UINT		:= 1;		(*Webserver enabled*)
END_VAR
